% RSLogix 500 project P3_BAK029.RSS, saved by version 8.30.00.16 %
PROJECT "UNTITLED"    % processor: Bul.1763 MicroLogix 1100 Series B %

PROGRAM FILES
  LAD 2 "MAIN"  9 rungs

DATA FILES
  O0 OUTPUT  4 elements
  I1 INPUT  6 elements
  S2 STATUS  66 elements
  B3 BINARY  2 elements
  T4 TIMER  1 elements
  C5 COUNTER  1 elements
  R6 CONTROL  1 elements
  N7 INTEGER  9 elements
  F8 FLOAT  1 elements
  ST9 STRING  10 elements

LADDER 2 "MAIN"
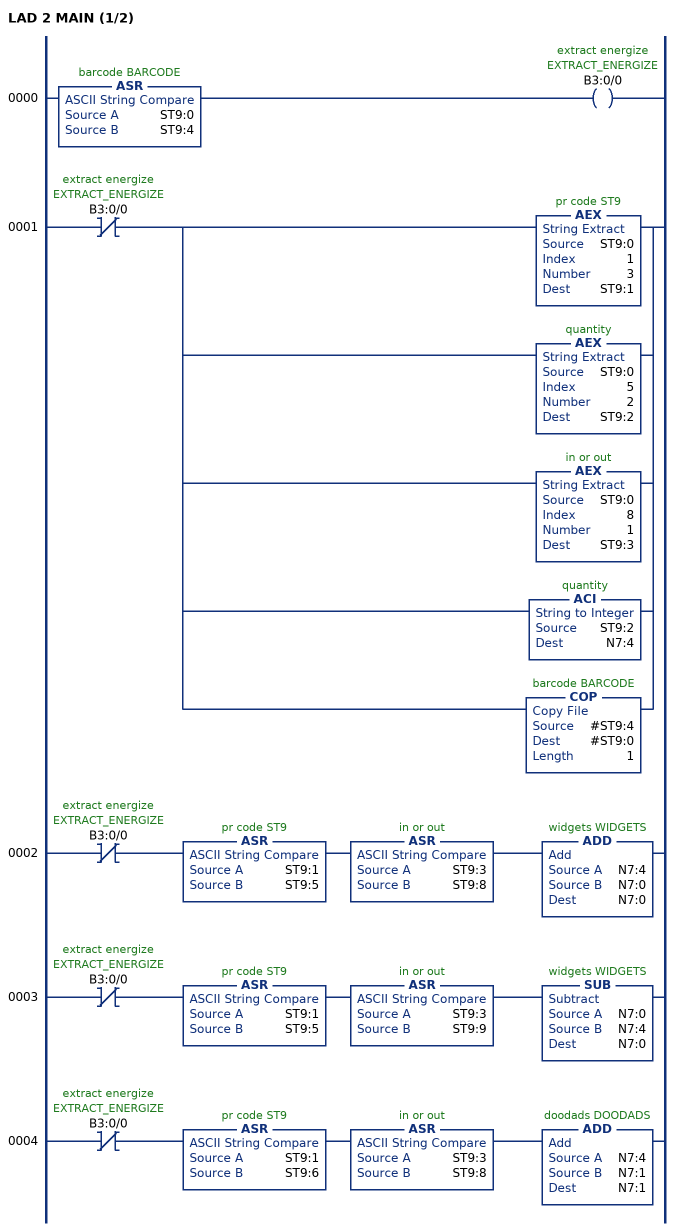
% Rung: 0 %
SOR ASR ST9:0 ST9:4 OTE B3:0/0 EOR
%   ST9:0  BARCODE  "barcode" %
%   ST9:4  "zero value" %
%   B3:0/0  EXTRACT_ENERGIZE  "extract energize" %
% Rung: 1 %
SOR XIO B3:0/0 BST AEX ST9:0 1 3 ST9:1 NXB AEX ST9:0 5 2 ST9:2 NXB AEX ST9:0 8 1 ST9:3 NXB ACI ST9:2 N7:4 NXB COP #ST9:4 #ST9:0 1 BND EOR
%   B3:0/0  EXTRACT_ENERGIZE  "extract energize" %
%   ST9:0  BARCODE  "barcode" %
%   ST9:1  ST9  "pr code" %
%   ST9:2  "quantity" %
%   ST9:3  "in or out" %
%   N7:4  "quantity" %
%   ST9:4  "zero value" %
% Rung: 2 %
SOR XIO B3:0/0 ASR ST9:1 ST9:5 ASR ST9:3 ST9:8 ADD N7:4 N7:0 N7:0 EOR
%   B3:0/0  EXTRACT_ENERGIZE  "extract energize" %
%   ST9:1  ST9  "pr code" %
%   ST9:5  "zero value" %
%   ST9:3  "in or out" %
%   ST9:8  "incoming" %
%   N7:4  "quantity" %
%   N7:0  WIDGETS  "widgets" %
% Rung: 3 %
SOR XIO B3:0/0 ASR ST9:1 ST9:5 ASR ST9:3 ST9:9 SUB N7:0 N7:4 N7:0 EOR
%   B3:0/0  EXTRACT_ENERGIZE  "extract energize" %
%   ST9:1  ST9  "pr code" %
%   ST9:5  "zero value" %
%   ST9:3  "in or out" %
%   ST9:9  "outgoing" %
%   N7:0  WIDGETS  "widgets" %
%   N7:4  "quantity" %
% Rung: 4 %
SOR XIO B3:0/0 ASR ST9:1 ST9:6 ASR ST9:3 ST9:8 ADD N7:4 N7:1 N7:1 EOR
%   B3:0/0  EXTRACT_ENERGIZE  "extract energize" %
%   ST9:1  ST9  "pr code" %
%   ST9:6  "doodads" %
%   ST9:3  "in or out" %
%   ST9:8  "incoming" %
%   N7:4  "quantity" %
%   N7:1  DOODADS  "doodads" %

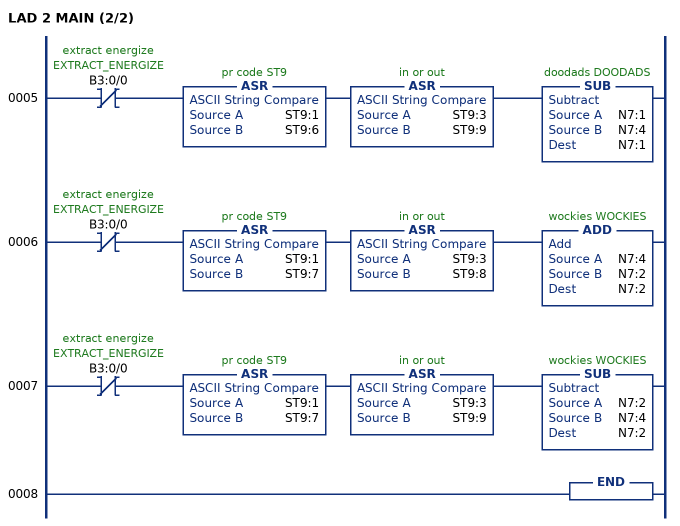
% Rung: 5 %
SOR XIO B3:0/0 ASR ST9:1 ST9:6 ASR ST9:3 ST9:9 SUB N7:1 N7:4 N7:1 EOR
%   B3:0/0  EXTRACT_ENERGIZE  "extract energize" %
%   ST9:1  ST9  "pr code" %
%   ST9:6  "doodads" %
%   ST9:3  "in or out" %
%   ST9:9  "outgoing" %
%   N7:1  DOODADS  "doodads" %
%   N7:4  "quantity" %
% Rung: 6 %
SOR XIO B3:0/0 ASR ST9:1 ST9:7 ASR ST9:3 ST9:8 ADD N7:4 N7:2 N7:2 EOR
%   B3:0/0  EXTRACT_ENERGIZE  "extract energize" %
%   ST9:1  ST9  "pr code" %
%   ST9:7  "wockies" %
%   ST9:3  "in or out" %
%   ST9:8  "incoming" %
%   N7:4  "quantity" %
%   N7:2  WOCKIES  "wockies" %
% Rung: 7 %
SOR XIO B3:0/0 ASR ST9:1 ST9:7 ASR ST9:3 ST9:9 SUB N7:2 N7:4 N7:2 EOR
%   B3:0/0  EXTRACT_ENERGIZE  "extract energize" %
%   ST9:1  ST9  "pr code" %
%   ST9:7  "wockies" %
%   ST9:3  "in or out" %
%   ST9:9  "outgoing" %
%   N7:2  WOCKIES  "wockies" %
%   N7:4  "quantity" %
% Rung: 8 %
SOR END EOR

OTHER DOCUMENTED ADDRESSES
  B3:0/5  "ons"
  B3:0/6  "ons"
  B3:0/7  "ons"
  B3:0/8  "ons"
  B3:0/9  "ons"
  B3:0/10  "0ns"
  B3:0/11  "ons"
  B3:1/0  "ons"
  B3:1/1  "ons"
  B3:1/2  "ons"
  B3:1/3  "ons"
  B3:1/4  "ons"
  B3:1/5  "o"
  B3:1/6  "o"
  B3:1/7  "0"
  N7:3  ST  "product index"
  N7:5  "in or out num"
  N7:6  "yyy"
  N7:8  "zero value"
  PFILE:4  "controls"
  R6:0  "barcode"
  ST9:0.0  "length"
  ST9:1.0  "pr"
  ST9:2.0  "qq"
  ST9:3.0  "in/out"
  ST9:4.0  "compare"
  U:3  "i/o"
  U:4  "controls"

DATA TABLE (non-zero values as saved)
DATA B3
% B3:0 % 0X0040 0X0000
DATA ST9
% ST9:5 % "123"
% ST9:6 % "456"
% ST9:7 % "789"
% ST9:8 % "1"
% ST9:9 % "2"
